FUNCTION MILLIARCSEC_TO_DEG : LREAL
VAR_INPUT
    mas : LREAL;
END_VAR
VAR
END_VAR

MILLIARCSEC_TO_DEG := mas / 3600000.0;

END_FUNCTION

(* stored: Version 1.1.0.1, ProductVersion 3.1.4018.5
   POU MILLIARCSEC_TO_DEG: Id {1dc291b7-6302-4dd4-a419-fb710d7fe088}, SpecialFunc None *)
